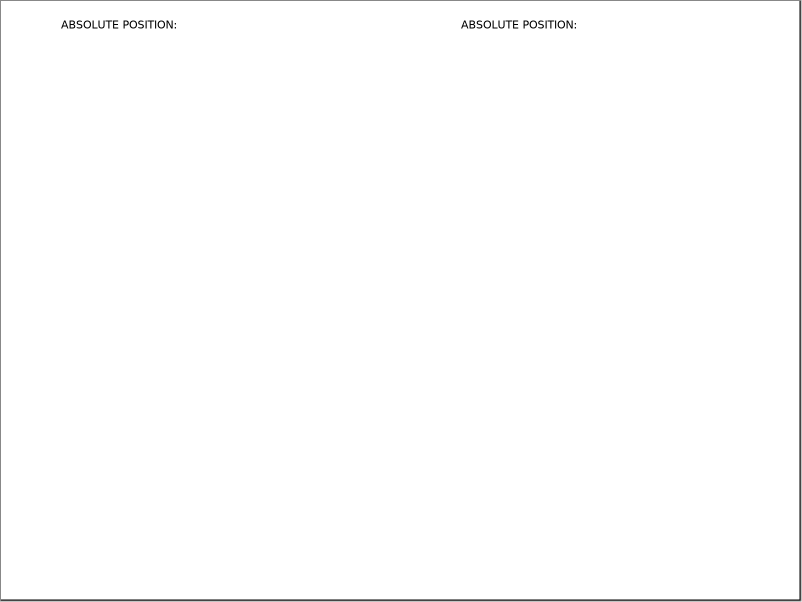
VISUALIZATION F45_Phasing_Absolute  // 802x602
    Rectangle (0,0 800x600)
    Label (10,10 170x30), "ABSOLUTE POSITION:"
    Label (410,10 170x30), "ABSOLUTE POSITION:"
END_VISUALIZATION

(* stored: Version 1.1.0.1, ProductVersion 3.1.4022.7
   Visu F45_Phasing_Absolute: Id {a7fcd5b7-675d-4d65-8554-ce917ee697cc} *)
